// TIA Portal V16 program export: 1 tag tables, 0 data types, 0 data blocks, 1 code blocks (in call order from the OBs), 1 instance data blocks

VAR_GLOBAL   // PLC tag table "Automatic_Gate_Example"
   stop AT %I0.0 : Bool;
   overcurrent_relay AT %I0.1 : Bool;
   system AT %M0.0 : Bool;
   up_directon_sensor AT %I0.5 : Bool;
   down_direction_sensor AT %I0.4 : Bool;
   open_limit AT %I0.2 : Bool;
   close_limit AT %I0.3 : Bool;
   open_gate AT %Q0.0 : Bool;
   close_gate AT %Q0.1 : Bool;
   gate_time AT %M0.1 : Bool;
END_VAR

ORGANIZATION_BLOCK "Automatic_Gate_Example"   // OB1, LAD, ProgramCycle
TITLE = "Main Program Sweep (Cycle)"
{ S7_Optimized_Access := 'TRUE' }
VERSION : 0.1
// stored: AutoNumber true, IsIECCheckEnabled false, SetENOAutomatically false
   VAR_INPUT
      Initial_Call : Bool;   // Initial call of this OB
      Remanence : Bool;   // =True, if remanent data are available
   END_VAR
BEGIN

REGION Network 1
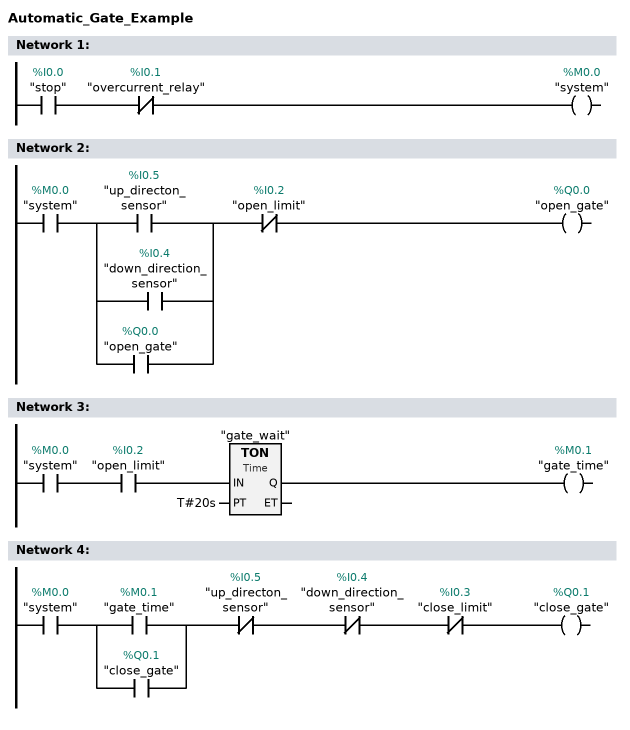
   RUNG wire#powerrail
      Contact( "stop" )
      I_Contact( "overcurrent_relay" )
      Coil( "system" )
   END_RUNG
   // the same network as SCL:
   "system" := "stop" AND NOT "overcurrent_relay";
END_REGION

REGION Network 2
   RUNG wire#powerrail
      Contact( "system" )
      wire#w1
      Contact( "up_directon_sensor" )
      wire#w2
      I_Contact( "open_limit" )
      Coil( "open_gate" )
   END_RUNG
   RUNG wire#w1
      Contact( "down_direction_sensor" )
   END_RUNG wire#w2
   RUNG wire#w1
      Contact( "open_gate" )
   END_RUNG wire#w2
   // the same network as SCL:
   "open_gate" := "system" AND ("up_directon_sensor" OR "down_direction_sensor" OR "open_gate") AND NOT "open_limit";
END_REGION

REGION Network 3
   RUNG wire#powerrail
      Contact( "system" )
      Contact( "open_limit" )
      { S7_Templates := "time_type := Time" } "gate_wait".TON(pt := T#20s, et =>)
      Coil( "gate_time" )
   END_RUNG
   // the same network as SCL:
   "gate_wait".TON(IN := "system" AND "open_limit", PT := T#20s);
   "gate_time" := "gate_wait".Q;
END_REGION

REGION Network 4
   RUNG wire#powerrail
      Contact( "system" )
      wire#w1
      Contact( "gate_time" )
      wire#w2
      I_Contact( "up_directon_sensor" )
      I_Contact( "down_direction_sensor" )
      I_Contact( "close_limit" )
      Coil( "close_gate" )
   END_RUNG
   RUNG wire#w1
      Contact( "close_gate" )
   END_RUNG wire#w2
   // the same network as SCL:
   "close_gate" := "system" AND ("gate_time" OR "close_gate") AND NOT "up_directon_sensor" AND NOT "down_direction_sensor" AND NOT "close_limit";
END_REGION
END_ORGANIZATION_BLOCK

DATA_BLOCK "gate_wait"   // DB2
{ S7_Optimized_Access := 'TRUE' }
// stored: AutoNumber true, DBAccessibleFromOPCUA true, InstanceOfName IEC_TIMER, OfSystemLibElement IEC_TIMER, OfSystemLibVersion 1.0
"IEC_TIMER"
   // VAR
   //    PT : Time;
   //    ET { ExternalWritable := 'False'} : Time;
   //    IN : Bool;
   //    Q { ExternalWritable := 'False'} : Bool;
   // END_VAR
BEGIN
END_DATA_BLOCK
